(****************************************************************************************)
(*							Beckhoff Automation Poland									*)
(*								FB_GetSystemTime  v1.2									*)
(*									26.07.2013											*)
(*		v1.2 - zmiana nazwy bloku z FB_Time na FB_GetSystemTime, dodanie wyjscia DT		*)
(*		v1.1 - dodano na wyjściu zmienną czasu w formie struktury TIMESTRUCT 			*)
(*				Blok funkcyjny podający dokładną datę w odrębnych zmiennych				*)
(*						może być wywołany raz w programie PLC							*)
(*						Wymaga dodania biblioteki TcUtilities.lib						*)
(*______________________________________________________________________________________*)
FUNCTION_BLOCK FB_GetSystemTime
VAR_INPUT
	bEnable:			BOOL;				(*Aktywuje pobieranie czasu systemowego*)
END_VAR
VAR_OUTPUT
	stActTime			:	TIMESTRUCT;
	dtActTime: DT;
(*Poszczególne składowe daty*)
	wYear 				:	WORD;
	wMonth 				:	WORD;
	wDayOfWeek 			: 	WORD;
	wDay 				:	WORD;
	wHour 				:	WORD;
	wMinute 			:	WORD;
	wSecond 			:	WORD;
	wMilliseconds 		: 	WORD;
END_VAR
VAR
	fbGetTime			:	NT_GetTime;
	Get					:	TON;
END_VAR
VAR CONSTANT
	tFrequency			:	TIME			:= T#1s;				(*Częstotliwość pobierania czasu*)
END_VAR

Get(IN:= NOT Get.Q AND bEnable, PT:=tFrequency);
fbGetTime(
	NETID:= '',
	START:= Get.Q,
	TMOUT:= T#200ms,
	TIMESTR=>stActTime);

dtActTime 		:= SYSTEMTIME_TO_DT(stActTime);
wDay 			:= stActTime.wDay;
wDayOfWeek 		:= stActTime.wDayOfWeek;
wHour 			:= stActTime.wHour;
wMilliseconds 	:= stActTime.wMilliseconds;
wMinute 		:= stActTime.wMinute;
wMonth 			:= stActTime.wMonth;
wSecond 		:= stActTime.wSecond;
wYear 			:= stActTime.wYear;

END_FUNCTION_BLOCK

(* stored: Version 1.1.0.1, ProductVersion 3.1.4026.13, FileIdentifier a948dc312669a5a7e0544cb3a703a54b5d2ef1a9, FileSignature 2a81768b7118fe0dc39a846adcda4d4a3b54b6c67885d4c3d2489cd789f604faf2463e03f988b8b2b0ac8dd13ef6ecfe71adda54b37a4fabc69be48f653288715a1c280680a498b731465dfa1b0d280e12f894314a2586d7e585e667f0c213658f7a45338fc80483d7e2974365d9ecef360ae11f2d42fbefb4c37799d35095f5d275a767d77e557cb328d484a58f2b15ece7812567923b3ac3169efab73e7b2fb8048e15d0494c9ec42455702cfd45bc853b7ab5a9a9b803833766d2c407092514d5f731621fdc243b18f35b37ade55ebd4339f460898501ea385adc83164e823e6beb94c1df003afacc83815cbd689357e27594ffc49c22745b9ab309401dcd
   POU FB_GetSystemTime: Id {51eef71f-6694-4d65-ad0d-61201ea67dc9}, SpecialFunc None *)
